{attribute addProperty BoxType "EK1100-0000-0018"}
{attribute addProperty Id "Beckhoff_EJ7xxxEK1122Beckhoff_EJ7xxxEK1122_22994AD2162A_0001_EJ7031_0000_0026EJ7031_26D8313822628.25A_0002_EJ7037_0000_0020EJ7037_F30AD12822628.25A_0003_EJ7041_0052_0016EJ7041_26D8313822628.25A_0004_EJ7047_0000_0018EJ7047_F30AD12822628.25A_0005_EJ7047_0000_0019EJ7047_F30AD12822628.25A_0006_EJ7047_0000_0020EJ7047_F30AD12822628.25A_0007_EJ7342_0000_0019EJ7342_E03DC37137046.25A_0008_EJ7342_0000_0020EJ7342_E2585B8337046.25A_0009_EJ7211_0010_0026EJ7211_83D4128E25031.25A_0010_EJ7211_0010_0027EJ7211_83D4128E25031.25A_0011_EJ7211_0010_0028EJ7211_83D4128E25031.25A_0012_EJ7211_0010_0029EJ7211_83D4128E25031.25A_0013_EJ7211_0010_0030EJ7211_2D7B43DC25832.25A_0014_EJ7211_0010_0031EJ7211_2D7B43DC25832.25A_0015_EJ7211_0010_0032EJ7211_2D7B43DC25832.25A_0016_EJ7211_0011_0026EJ7211_789C0F5925031.25A_0017_EJ7211_0011_0027EJ7211_789C0F5925031.25A_0018_EJ7211_0011_0028EJ7211_789C0F5925031.25A_0019_EJ7211_0011_0029EJ7211_789C0F5925031.25A_0020_EJ7211_0011_0030EJ7211_789C0F5925031.25A_0021_EJ7211_0011_0031EJ7211_789C0F5925031.25A_0022_EJ7211_0011_0032EJ7211_789C0F5925031.25A_0023_EJ7211_9414_0029EJ7211_83D4128E25031.25A_0024_EJ7211_9414_0030EJ7211_5D87091826633.25A_0025_EJ7211_9414_0031EJ7211_5D87091826633.25A_0026_EJ7211_9414_0032EJ7211_5D87091826633.25A_0027_EJ7211_9415_0029EJ7211_789C0F5925031.25A_0028_EJ7211_9415_0030EJ7211_789C0F5925031.25A_0029_EJ7211_9415_0031EJ7211_789C0F5925031.25A_0030_EJ7211_9415_0032EJ7211_789C0F5925031.25A_0031_EJ7334_0008_0016EJ7334_68079CA927434.25A_0032_EJ7411_0000_0018EJ7411_675FBD0529036.25"}
{attribute addProperty CRC "2675245358"}
{attribute addProperty SizeInBites "8248"}
{attribute addProperty SizeInBytes "1031"}
TYPE Beckhoff_EJ7xxx_9F75012E EXTENDS EK1100_179A0949 :
STRUCT
	{attribute addProperty Name "Beckhoff_EJ7xxxEK1122"}
	Beckhoff_EJ7xxxEK1122 : Beckhoff_EJ7xxxEK1122_22994AD2;
	{attribute addProperty Name "A_0001_EJ7031_0000_0026"}
	A_0001_EJ7031_0000_0026 : EJ7031_26D83138;
	{attribute addProperty Name "A_0002_EJ7037_0000_0020"}
	A_0002_EJ7037_0000_0020 : EJ7037_F30AD128;
	{attribute addProperty Name "A_0003_EJ7041_0052_0016"}
	A_0003_EJ7041_0052_0016 : EJ7041_26D83138;
	{attribute addProperty Name "A_0004_EJ7047_0000_0018"}
	A_0004_EJ7047_0000_0018 : EJ7047_F30AD128;
	{attribute addProperty Name "A_0005_EJ7047_0000_0019"}
	A_0005_EJ7047_0000_0019 : EJ7047_F30AD128;
	{attribute addProperty Name "A_0006_EJ7047_0000_0020"}
	A_0006_EJ7047_0000_0020 : EJ7047_F30AD128;
	{attribute addProperty Name "A_0007_EJ7342_0000_0019"}
	A_0007_EJ7342_0000_0019 : EJ7342_E03DC371;
	{attribute addProperty Name "A_0008_EJ7342_0000_0020"}
	A_0008_EJ7342_0000_0020 : EJ7342_E2585B83;
	{attribute addProperty Name "A_0009_EJ7211_0010_0026"}
	A_0009_EJ7211_0010_0026 : EJ7211_83D4128E;
	{attribute addProperty Name "A_0010_EJ7211_0010_0027"}
	A_0010_EJ7211_0010_0027 : EJ7211_83D4128E;
	{attribute addProperty Name "A_0011_EJ7211_0010_0028"}
	A_0011_EJ7211_0010_0028 : EJ7211_83D4128E;
	{attribute addProperty Name "A_0012_EJ7211_0010_0029"}
	A_0012_EJ7211_0010_0029 : EJ7211_83D4128E;
	{attribute addProperty Name "A_0013_EJ7211_0010_0030"}
	A_0013_EJ7211_0010_0030 : EJ7211_2D7B43DC;
	{attribute addProperty Name "A_0014_EJ7211_0010_0031"}
	A_0014_EJ7211_0010_0031 : EJ7211_2D7B43DC;
	{attribute addProperty Name "A_0015_EJ7211_0010_0032"}
	A_0015_EJ7211_0010_0032 : EJ7211_2D7B43DC;
	{attribute addProperty Name "A_0016_EJ7211_0011_0026"}
	A_0016_EJ7211_0011_0026 : EJ7211_789C0F59;
	{attribute addProperty Name "A_0017_EJ7211_0011_0027"}
	A_0017_EJ7211_0011_0027 : EJ7211_789C0F59;
	{attribute addProperty Name "A_0018_EJ7211_0011_0028"}
	A_0018_EJ7211_0011_0028 : EJ7211_789C0F59;
	{attribute addProperty Name "A_0019_EJ7211_0011_0029"}
	A_0019_EJ7211_0011_0029 : EJ7211_789C0F59;
	{attribute addProperty Name "A_0020_EJ7211_0011_0030"}
	A_0020_EJ7211_0011_0030 : EJ7211_789C0F59;
	{attribute addProperty Name "A_0021_EJ7211_0011_0031"}
	A_0021_EJ7211_0011_0031 : EJ7211_789C0F59;
	{attribute addProperty Name "A_0022_EJ7211_0011_0032"}
	A_0022_EJ7211_0011_0032 : EJ7211_789C0F59;
	{attribute addProperty Name "A_0023_EJ7211_9414_0029"}
	A_0023_EJ7211_9414_0029 : EJ7211_83D4128E;
	{attribute addProperty Name "A_0024_EJ7211_9414_0030"}
	A_0024_EJ7211_9414_0030 : EJ7211_5D870918;
	{attribute addProperty Name "A_0025_EJ7211_9414_0031"}
	A_0025_EJ7211_9414_0031 : EJ7211_5D870918;
	{attribute addProperty Name "A_0026_EJ7211_9414_0032"}
	A_0026_EJ7211_9414_0032 : EJ7211_5D870918;
	{attribute addProperty Name "A_0027_EJ7211_9415_0029"}
	A_0027_EJ7211_9415_0029 : EJ7211_789C0F59;
	{attribute addProperty Name "A_0028_EJ7211_9415_0030"}
	A_0028_EJ7211_9415_0030 : EJ7211_789C0F59;
	{attribute addProperty Name "A_0029_EJ7211_9415_0031"}
	A_0029_EJ7211_9415_0031 : EJ7211_789C0F59;
	{attribute addProperty Name "A_0030_EJ7211_9415_0032"}
	A_0030_EJ7211_9415_0032 : EJ7211_789C0F59;
	{attribute addProperty Name "A_0031_EJ7334_0008_0016"}
	A_0031_EJ7334_0008_0016 : EJ7334_68079CA9;
	{attribute addProperty Name "A_0032_EJ7411_0000_0018"}
	A_0032_EJ7411_0000_0018 : EJ7411_675FBD05;
END_STRUCT
END_TYPE

(* stored: Version 1.2.0.0, ProductVersion 3.1.4024.9
   DUT Beckhoff_EJ7xxx_9F75012E: Id {414b577b-820e-4719-b999-416d32fa9237} *)
